// TwinCAT 3 PLC project PLC
// ProgramVersion: 3.1.4023.0
// libraries:
//   EfficientIO Communicator, * (EfficientIO)
//   EfficientIO ModbusTCP, * (EfficientIO)
//   Lynus Energy Basic, * (Lynus AG)
//   Lynus Persistent Data V1, * (Lynus AG)
//   Lynus Standards, * (Lynus AG)
//   Tc2_IoFunctions, * (Beckhoff Automation GmbH)
//   Tc2_ModbusRTU, * (Beckhoff Automation GmbH)
//   Tc2_ModbusSrv, * (Beckhoff Automation GmbH)
//   Tc2_SerialCom, * (Beckhoff Automation GmbH)
//   Tc2_Standard, * (Beckhoff Automation GmbH)
//   Tc2_System, * (Beckhoff Automation GmbH)
//   Tc2_Utilities, * (Beckhoff Automation GmbH)
//   Tc3_IotBase, * (Beckhoff Automation GmbH)
//   Tc3_Module, * (Beckhoff Automation GmbH)
// project tree:
//   DUTs/ ModbusRTURequest.TcDUT (not stored), struct_ADS_Barac.TcDUT (not stored)
//   / FastTask.TcTTO, MiddleTask.TcTTO, SlowTask.TcTTO
//   FB/ F_Convert_Reg_to_Real.TcPOU, MODBUS_RTU_Olymp.TcPOU
//   POUs/ prgBattery.TcPOU, prgComEffIO.TcPOU, prgCS.TcPOU, prgEM.TcPOU, prgEMS.TcPOU, prgHeatPump.TcPOU, prgPersistent.TcPOU, prgPV.TcPOU, prgRWEffIO.TcPOU (not stored), prgTemperature.TcPOU, prgVarEffIO.TcPOU
// real-time tasks:
//   TASK PlcTask: cycle T#10ms, priority 20, ADS port 350
//   TASK FastTask: cycle T#5ms, priority 19, ADS port 351
//   TASK MiddleTask: cycle T#10ms, priority 21, ADS port 352
//   TASK SlowTask: cycle T#20ms, priority 22, ADS port 353
// I/O:
//   DEVICE Gerät 2 (CX-BK)
//     Box 1 (CX-BK)
// variable links:
//   PLC/PLC Instance <-> Device 2 (CX-BK)/Box 1 (CX-BK)
//     FastTask Inputs/MODBUS_RTU_Olymp.fbModbusRtuMaster_KL6x22B.InData/D[{0..21}] <-> Term 6 (KL6041)/Channel 1/Data In {0..21}  (22 links)
//     FastTask Inputs/MODBUS_RTU_Olymp.fbModbusRtuMaster_KL6x22B.InData/Status <-> Term 6 (KL6041)/Channel 1/Status
//     FastTask Outputs/MODBUS_RTU_Olymp.fbModbusRtuMaster_KL6x22B.OutData/Ctrl <-> Term 6 (KL6041)/Channel 1/Ctrl
//     FastTask Outputs/MODBUS_RTU_Olymp.fbModbusRtuMaster_KL6x22B.OutData/D[{0..21}] <-> Term 6 (KL6041)/Channel 1/Data Out {0..21}  (22 links)
//     MiddleTask Inputs/prgEM.fbEM1.fbKL3403.byStateCH1 <-> Term 5 (KL3403)/Channel 1/Status
//     MiddleTask Inputs/prgEM.fbEM1.fbKL3403.byStateCH2 <-> Term 5 (KL3403)/Channel 2/Status
//     MiddleTask Inputs/prgEM.fbEM1.fbKL3403.byStateCH3 <-> Term 5 (KL3403)/Channel 3/Status
//     MiddleTask Inputs/prgEM.fbEM1.fbKL3403.iDataInCH1 <-> Term 5 (KL3403)/Channel 1/Daten Ein
//     MiddleTask Inputs/prgEM.fbEM1.fbKL3403.iDataInCH2 <-> Term 5 (KL3403)/Channel 2/Daten Ein
//     MiddleTask Inputs/prgEM.fbEM1.fbKL3403.iDataInCH3 <-> Term 5 (KL3403)/Channel 3/Daten Ein
//     MiddleTask Inputs/prgEM.fbKBusState.uiKBusState_OUT <-> Inputs/State
//     MiddleTask Inputs/prgTemperature.stInData_1/iDataIn <-> Term 4 (KL3204)/Channel 1/Daten Ein
//     MiddleTask Inputs/prgTemperature.stInData_2/iDataIn <-> Term 4 (KL3204)/Channel 2/Daten Ein
//     MiddleTask Inputs/prgTemperature.stInData_1/iState <-> Term 4 (KL3204)/Channel 1/Status
//     MiddleTask Inputs/prgTemperature.stInData_2/iState <-> Term 4 (KL3204)/Channel 2/Status
//     MiddleTask Outputs/prgEM.fbEM1.fbKL3403.byCntrCH1 <-> Term 5 (KL3403)/Channel 1/Kontrolle
//     MiddleTask Outputs/prgEM.fbEM1.fbKL3403.byCntrCH2 <-> Term 5 (KL3403)/Channel 2/Kontrolle
//     MiddleTask Outputs/prgEM.fbEM1.fbKL3403.byCntrCH3 <-> Term 5 (KL3403)/Channel 3/Kontrolle
//     MiddleTask Outputs/prgTemperature.bout_Boiler1_6kW <-> Term 3 (KL2408)/Channel 1/Ausgang
//     MiddleTask Outputs/prgTemperature.bout_Boiler2_10kW <-> Term 3 (KL2408)/Channel 2/Ausgang
//     MiddleTask Outputs/prgTemperature.stOutData_1/iCtrl <-> Term 4 (KL3204)/Channel 1/Kontrolle
//     MiddleTask Outputs/prgTemperature.stOutData_2/iCtrl <-> Term 4 (KL3204)/Channel 2/Kontrolle
//     MiddleTask Outputs/prgTemperature.stOutData_1/iDataOut <-> Term 4 (KL3204)/Channel 1/Daten Aus
//     MiddleTask Outputs/prgTemperature.stOutData_2/iDataOut <-> Term 4 (KL3204)/Channel 2/Daten Aus

CONFIGURATION PLC
    RESOURCE PLC ON TwinCAT3
        TASK FastTask(INTERVAL := T#5ms, PRIORITY := 19);
        TASK MiddleTask(INTERVAL := T#10ms, PRIORITY := 21);
        TASK SlowTask(INTERVAL := T#20ms, PRIORITY := 22);
        PROGRAM prgVarEffIO WITH FastTask : prgVarEffIO;
        PROGRAM prgRWEffIO WITH FastTask : prgRWEffIO;
        PROGRAM prgHeatPump WITH FastTask : prgHeatPump;
        PROGRAM prgEM WITH MiddleTask : prgEM;
        PROGRAM prgTemperature WITH MiddleTask : prgTemperature;
        PROGRAM prgPV WITH MiddleTask : prgPV;
        PROGRAM prgBattery WITH MiddleTask : prgBattery;
        PROGRAM prgEMS WITH MiddleTask : prgEMS;
        PROGRAM prgPersistent WITH MiddleTask : prgPersistent;
        PROGRAM prgCS WITH MiddleTask : prgCS;
        PROGRAM prgComEffIO WITH SlowTask : prgComEffIO;
    END_RESOURCE
END_CONFIGURATION

// ---- POUs/prgVarEffIO.TcPOU
PROGRAM prgVarEffIO
VAR
	fbVar		: FB_VarInfo_V3;
END_VAR

fbVar(
	bReadInfo:= , 
	eTMCFile:= eSelectTMCFile.eDontUseTMCFile, 
	eSavePositionTMCFile:= eSavePositionOnPLC.ePostionHardDisk, 
	udiCounterFoundVariables=> , 
	bError=> , 
	bBusy=> , 
	byProgress=> , 
	udiErrorCodeOut=> , 
	eErrorVarInfo_Out=> , 
	sVarWithError=> );

fbVar(
	bReadInfo:= , 
	eTMCFile:= eSelectTMCFile.eDontUseTMCFile, 
	eSavePositionTMCFile:= eSavePositionOnPLC.ePostionHardDisk, 
	udiCounterFoundVariables=> , 
	bError=> , 
	bBusy=> , 
	byProgress=> , 
	udiErrorCodeOut=> , 
	eErrorVarInfo_Out=> , 
	sVarWithError=> );
	
fbVar(
	bReadInfo:= , 
	eTMCFile:= eSelectTMCFile.eDontUseTMCFile, 
	eSavePositionTMCFile:= eSavePositionOnPLC.ePostionHardDisk, 
	udiCounterFoundVariables=> , 
	bError=> , 
	bBusy=> , 
	byProgress=> , 
	udiErrorCodeOut=> , 
	eErrorVarInfo_Out=> , 
	sVarWithError=> );

END_PROGRAM

// ---- POUs/prgHeatPump.TcPOU
PROGRAM prgHeatPump
VAR
	byte_OperationMode_H1: BYTE;							//{#lynus.ag#()}
	real_ComfortSetpoint_H1 :REAL;							//{#lynus.ag#()}
	real_ReducedSetpoint_H1: REAL;							//{#lynus.ag#()}
	real_HeatingCurveSlope_H1:REAL;							//{#lynus.ag#()}
	real_HeatingCurveDisplacement_H1: REAL;					//{#lynus.ag#()}
	real_RelativeRoomHumidity1_H1: REAL;	
	real_RoomTemperature1_H1 : REAL;
	real_RoomSetpoint1_H1 : REAL;
	real_FlowTemperature1_H1 : REAL;						//{#lynus.ag#()}
	real_FlowTemperatureSetpoint1_H1 : REAL;				//{#lynus.ag#()}
	m_RoomThermostat1_H1 : BOOL;							//{#lynus.ag#()}
	real_HeatOutput :REAL;									//{#lynus.ag#()}
	real_HeatInputSource :REAL;								//{#lynus.ag#()}
	real_PowerConsumption :REAL;							//{#lynus.ag#()}
	m_Heatingcircuit1_H1 : BOOL;							//{#lynus.ag#()}
	FB_DwordToWord :FB_CV_WORD_TO_DWORD;

	real_Outside_Temp : REAL;								//{#lynus.ag#()}
	real_Outside_Temp_min : REAL;							//{#lynus.ag#()}
	real_Outside_Temp_max : REAL;							//{#lynus.ag#()}
	real_Outside_Temp_attenuated : REAL;					//{#lynus.ag#()}
	real_Outside_Temp_composite : REAL;						//{#lynus.ag#()}

END_VAR

MODBUS_RTU_Olymp();

byte_OperationMode_H1 		:= 	WORD_TO_BYTE(Modbus_RTU_Olymp.structArrayModbusRTU[1].wArrayReceiveBuffer[0]);
real_ComfortSetpoint_H1		:= 	word_TO_REAL(Modbus_RTU_Olymp.structArrayModbusRTU[1].wArrayReceiveBuffer[1])/64;
real_ReducedSetpoint_H1		:= 	word_TO_REAL(Modbus_RTU_Olymp.structArrayModbusRTU[1].wArrayReceiveBuffer[2])/64;
real_HeatingCurveSlope_H1	:= 	WORD_TO_REAL(Modbus_RTU_Olymp.structArrayModbusRTU[1].wArrayReceiveBuffer[4])/50;
real_HeatingCurveDisplacement_H1:= 	WORD_TO_REAL(Modbus_RTU_Olymp.structArrayModbusRTU[1].wArrayReceiveBuffer[5])/64;
real_RelativeRoomHumidity1_H1:= 	word_TO_REAL(Modbus_RTU_Olymp.structArrayModbusRTU[1].wArrayReceiveBuffer[16])/1;
real_RoomTemperature1_H1	:= 	WORD_TO_REAL(Modbus_RTU_Olymp.structArrayModbusRTU[1].wArrayReceiveBuffer[18])/64;
real_RoomSetpoint1_H1		:= 	word_TO_REAL(Modbus_RTU_Olymp.structArrayModbusRTU[1].wArrayReceiveBuffer[20])/64;
real_FlowTemperature1_H1	:= 	word_TO_REAL(Modbus_RTU_Olymp.structArrayModbusRTU[2].wArrayReceiveBuffer[0])/64;
real_FlowTemperatureSetpoint1_H1:= 	WORD_TO_REAL(Modbus_RTU_Olymp.structArrayModbusRTU[2].wArrayReceiveBuffer[2])/64;
m_RoomThermostat1_H1		:= 	WORD_TO_BOOL(Modbus_RTU_Olymp.structArrayModbusRTU[2].wArrayReceiveBuffer[4]);
m_Heatingcircuit1_H1		:= 	WORD_TO_BOOL(Modbus_RTU_Olymp.structArrayModbusRTU[2].wArrayReceiveBuffer[9]);


FB_DwordToWord( 	wInputValue_1 := Modbus_RTU_Olymp.structArrayModbusRTU[5].wArrayReceiveBuffer[0],
					wInputValue_2 := Modbus_RTU_Olymp.structArrayModbusRTU[5].wArrayReceiveBuffer[1],
					eByteOrderForConvert :=,
					dwOutputValue =>);
real_HeatOutput				:= 	DWORD_TO_REAL(FB_DwordToWord.dwOutputValue)/100;

FB_DwordToWord( 	wInputValue_1 := Modbus_RTU_Olymp.structArrayModbusRTU[5].wArrayReceiveBuffer[3],
					wInputValue_2 := Modbus_RTU_Olymp.structArrayModbusRTU[5].wArrayReceiveBuffer[4],
					eByteOrderForConvert :=,
					dwOutputValue =>);
real_HeatInputSource			:= 	DWORD_TO_REAL(FB_DwordToWord.dwOutputValue)/100;
					
FB_DwordToWord( 	wInputValue_1 := Modbus_RTU_Olymp.structArrayModbusRTU[5].wArrayReceiveBuffer[6],
					wInputValue_2 := Modbus_RTU_Olymp.structArrayModbusRTU[5].wArrayReceiveBuffer[7],
					eByteOrderForConvert :=,
					dwOutputValue =>);
real_PowerConsumption			:= 	DWORD_TO_REAL(FB_DwordToWord.dwOutputValue)/100;



real_Outside_Temp 				:= INT_TO_REAL(WORD_TO_INT(Modbus_RTU_Olymp.structArrayModbusRTU[6].wArrayReceiveBuffer[4]))/64;
real_Outside_Temp_min			:= INT_TO_REAL(WORD_TO_INT(Modbus_RTU_Olymp.structArrayModbusRTU[6].wArrayReceiveBuffer[6]))/64;
real_Outside_Temp_max			:= INT_TO_REAL(WORD_TO_INT(Modbus_RTU_Olymp.structArrayModbusRTU[6].wArrayReceiveBuffer[7]))/64;
real_Outside_Temp_attenuated	:= INT_TO_REAL(WORD_TO_INT(Modbus_RTU_Olymp.structArrayModbusRTU[6].wArrayReceiveBuffer[8]))/64;
real_Outside_Temp_composite		:= INT_TO_REAL(WORD_TO_INT(Modbus_RTU_Olymp.structArrayModbusRTU[6].wArrayReceiveBuffer[9]))/64;

END_PROGRAM

// ---- FB/MODBUS_RTU_Olymp.TcPOU
PROGRAM MODBUS_RTU_Olymp

VAR_INPUT

END_VAR
VAR_OUTPUT
	dword_MB_Error		:ARRAY[1..3] OF DWORD;
END_VAR
VAR
//	fbModbusRtuMaster_KL6x22B: ModbusRtuMaster_KL6x22B;
	fbModbusRtuMaster_KL6x22B: ModbusRtuMasterV2_KL6x22B;
	fbConfigKL6041 : KL6Configuration;
	uintPollOrderCount: UINT;
	mBusy: BOOL;
	mError: BOOL;
	mStart: BOOL;
	udintMemoryDestAddress: UDINT;
	udintBytesReceived: UDINT;
	intState: INT:=0;
	timerT1: TON;
	timeWaitT1: TIME:=T#500MS;
	timeWaitT2: TIME:=T#500MS;
	timeNoRxTimeout:	TIME:=T#2S;
	timerT2: TON;

	fb_F_TRIG1: F_TRIG;
	timerTimeout: TON;
	mError_Rx: BOOL;
	udintErrorID: MODBUS_ERRORS;
	byteClientSlaveID: BYTE;
	uintNoOfWords: UINT;
	uintStartAddress: UINT;
	dw_Mask: DWORD;
	dw_Mask_Not: DWORD;
	uint_TestPollOrder: UINT;
	mTestMode: BOOL;
	mInit_Done: BOOL;
	
	structArrayModbusRTU	:ARRAY[1..60] OF ModbusRTURequest;
	uintMaxModbusRTUOrders: UINT;
	mExecute: BOOL;
	int_Handshake: ComHandshake_t:=4;
	mode: ComSerialLineMode_t:=3;
	byte_DataBits: BYTE:=8;
	i: UINT;
END_VAR

(*
The function block "ModbusRtuMaster_KL6x22B" has 22 bytes where it communicates with the plc
software. These 22 bytes have to be assigned to the hardware device (for example KL/EL6021) in the
system manager plus the control and status byte.
If devices with less then 22 bytes are used, the other function blocks have to be used (for 5 bytes for example).
*)

(*
IF fbModbusRtuMaster_KL6x22B.MBmaster.TimeoutTON.Q=TRUE AND mTimeOUT_Qold=FALSE THEN mTimeOUT_Q_Rising; END_IF
mTimeOUT_Qold:=fbModbusRtuMaster_KL6x22B.MBmaster.TimeoutTON.Q;
*)

fb_F_TRIG1(CLK:=mBusy);

CASE intState OF

0: 	(* reset the start bit *)
	mStart:=FALSE;
	IF mInit_Done AND NOT fbConfigKL6041.Busy THEN 
		intState:=10;
		mExecute:=FALSE;		
	ELSE
		INIT();
		mExecute:=TRUE;		// necessary to write the communication parameters to the KL terminal. only necessary once if the terminal is brand new
	END_IF
10:
	(* set next poll order *)
	uintPollOrderCount:=uintPollOrderCount+1; (* next slave *)
	WHILE NOT structArrayModbusRTU[uintPollOrderCount].mRequestActive DO
		uintPollOrderCount:=uintPollOrderCount+1; (* next slave *)
	END_WHILE
	
	(* trouble shooting *)
	IF mTestMode THEN
		uintPollOrderCount:=uint_TestPollOrder; (* next slave *)
	END_IF
	
	IF uintPollOrderCount > uintMaxModbusRTUOrders OR uintPollOrderCount<1 THEN
		uintPollOrderCount:=1;
	END_IF

	udintMemoryDestAddress:=ADR(structArrayModbusRTU[uintPollOrderCount].wArrayReceiveBuffer[0]);
	structArrayModbusRTU[uintPollOrderCount].udintBytesReceived:=0;
	mStart:=TRUE;
	timerTimeout.IN:=TRUE;
	intState:=20;

20: (* wait for busy falling or time out *)
	IF fb_F_TRIG1.Q OR timerTimeout.Q THEN

		(* check answer time *)
		structArrayModbusRTU[uintPollOrderCount].timeTimeForRequest:=timerTimeout.ET;

		(* reset timer *)
		timerTimeout.IN:=FALSE;

		(* reset start bit *)
		mStart:=FALSE;

		(* save number of bytes received *)
		structArrayModbusRTU[uintPollOrderCount].udintBytesReceived:=udintBytesReceived;
		udintBytesReceived:=0;

		(* Error Detection *)
		IF timerTimeout.Q THEN
			mError_Rx:=TRUE;
			structArrayModbusRTU[uintPollOrderCount].udintErrorID:=9998;
			structArrayModbusRTU[uintPollOrderCount].strErrorMessage:='Timeout';
		ELSIF structArrayModbusRTU[uintPollOrderCount].udintBytesReceived=0 AND structArrayModbusRTU[uintPollOrderCount].uintNoOfWords>0 THEN
			mError_Rx:=TRUE;
			structArrayModbusRTU[uintPollOrderCount].udintErrorID:=9999;
			structArrayModbusRTU[uintPollOrderCount].strErrorMessage:='0 bytes received';
		ELSIF fbModbusRtuMaster_KL6x22B.Error THEN
			mError_Rx:=TRUE;
			structArrayModbusRTU[uintPollOrderCount].udintErrorID:=udintErrorID;
//			structArrayModbusRTU[uintPollOrderCount].strErrorMessage:=F_ADSERRORTEXT(structArrayModbusRTU[uintPollOrderCount].udintErrorID);
		ELSE
			mError_Rx:=FALSE;
			structArrayModbusRTU[uintPollOrderCount].udintErrorID:=0;
			structArrayModbusRTU[uintPollOrderCount].strErrorMessage:='';
		END_IF


		IF mError_Rx THEN
			structArrayModbusRTU[uintPollOrderCount].udintCommErrorCounter:=structArrayModbusRTU[uintPollOrderCount].udintCommErrorCounter+1;
		ELSIF structArrayModbusRTU[uintPollOrderCount].udintBytesReceived>0 THEN (* Rev 3 *)
			structArrayModbusRTU[uintPollOrderCount].udintCommSuccessCounter:=structArrayModbusRTU[uintPollOrderCount].udintCommSuccessCounter+1;
		END_IF

		structArrayModbusRTU[uintPollOrderCount].timerOKTimer.IN:=NOT mError_Rx;
		structArrayModbusRTU[uintPollOrderCount].timerErrorTimer.IN:=mError_Rx;

		dw_Mask:=1;
		dw_Mask:=SHL(dw_Mask,(structArrayModbusRTU[uintPollOrderCount].intDeviceNumber));
		dw_Mask_Not:=NOT dw_Mask;
		
		IF structArrayModbusRTU[uintPollOrderCount].timerErrorTimer.Q THEN
			structArrayModbusRTU[uintPollOrderCount].mError:=TRUE;
			IF structArrayModbusRTU[uintPollOrderCount].intDeviceClass>=1 AND structArrayModbusRTU[uintPollOrderCount].intDeviceClass<=3 THEN
				dword_MB_Error[structArrayModbusRTU[uintPollOrderCount].intDeviceClass]:=dword_MB_Error[structArrayModbusRTU[uintPollOrderCount].intDeviceClass] OR dw_Mask;
			END_IF
		END_IF

		IF structArrayModbusRTU[uintPollOrderCount].timerOKTimer.Q THEN
			structArrayModbusRTU[uintPollOrderCount].mError:=FALSE;
			IF structArrayModbusRTU[uintPollOrderCount].intDeviceClass>=1 AND structArrayModbusRTU[uintPollOrderCount].intDeviceClass<=3 THEN
				dword_MB_Error[structArrayModbusRTU[uintPollOrderCount].intDeviceClass]:=dword_MB_Error[structArrayModbusRTU[uintPollOrderCount].intDeviceClass] AND dw_Mask_Not;
			END_IF
		END_IF

		(* clear buffer *)
		IF mError_Rx THEN
			MEMSET(destAddr:=udintMemoryDestAddress,fillByte:=0,130);
		END_IF

		(* set next state *)
		intState:=30;
	END_IF

30:		(* wait *)
		timerT1(IN:=TRUE);
		IF timerT1.Q THEN
			timerT1(IN:=FALSE);
			intState:=0; (* back to start *)
		END_IF

END_CASE

(* Timer calls *)
structArrayModbusRTU[uintPollOrderCount].timerErrorTimer(PT:=timeNoRxTimeout);
structArrayModbusRTU[uintPollOrderCount].timerOKTimer(PT:=T#2S);
timerT1(PT:=timeWaitT1);
timerT2(PT:=timeWaitT2);
timerTimeout(PT:=timeNoRxTimeout+timeWaitT1);


(* Timers *)
structArrayModbusRTU[uintPollOrderCount].timerErrorTimer.PT:=T#5S;
structArrayModbusRTU[uintPollOrderCount].timerOKTimer.PT:=T#5S;


//fbModbusRtuMaster_KL6x22B.ReadInputRegs(
fbModbusRtuMaster_KL6x22B.ReadRegs(
	UnitID:= structArrayModbusRTU[uintPollOrderCount].byteClientSlaveID, 
	Quantity:= structArrayModbusRTU[uintPollOrderCount].uintNoOfWords, 
	MBAddr:= structArrayModbusRTU[uintPollOrderCount].uintStartAddress , 
	cbLength:= 2*structArrayModbusRTU[uintPollOrderCount].uintNoOfWords,
	pMemoryAddr:= udintMemoryDestAddress, 
	AuxQuantity:= , 
	AuxMBAddr:= , 
	AuxcbLength:= , 
	pAuxMemoryAddr:= , 
	Execute:= mStart, 
	Timeout:= T#1S, 
	BUSY=> mBusy, 
	Error=> mError, 
	ErrorId=> udintErrorID, 
	cbRead=> udintBytesReceived);
	
(*fbModbusRtuMaster_KL6x22B.ReadRegs(
	UnitID		:=structArrayModbusRTU[uintPollOrderCount].byteClientSlaveID,
	Quantity	:=structArrayModbusRTU[uintPollOrderCount].uintNoOfWords,
	MBAddr		:=structArrayModbusRTU[uintPollOrderCount].uintStartAddress,
	cbLength	:=2*structArrayModbusRTU[uintPollOrderCount].uintNoOfWords,
	pMemoryAddr	:=udintMemoryDestAddress,
	Execute		:=mStart,
	Timeout		:=t#1s,
	BUSY		=>mBusy,
	Error		=>mError,
	ErrorId		=>udintErrorID,
	cbRead		=>udintBytesReceived
);
*)
(*
(*fbModbusRtuMaster_KL6x22B.ReadInputRegs(
*)
fbModbusRtuMaster_KL6x22B.ReadInputRegs(
	UnitID		:=structArrayModbusRTU[uintPollOrderCount].byteClientSlaveID,
	Quantity	:=structArrayModbusRTU[uintPollOrderCount].uintNoOfWords,
	MBAddr		:=structArrayModbusRTU[uintPollOrderCount].uintStartAddress,
	cbLength	:=2*structArrayModbusRTU[uintPollOrderCount].uintNoOfWords,
	pMemoryAddr	:=udintMemoryDestAddress,
	Execute		:=mStart,
	Timeout		:=t#1s,
	BUSY		=>mBusy,
	Error		=>mError,
	ErrorId		=>udintErrorID,
	cbRead		=>udintBytesReceived
);
*)
// necessary for KL6041 to wirte the com settings
fbConfigKL6041(
	Execute 		:= mExecute,
	Mode 			:= mode,
	Baudrate 		:= 19200,
	NoDatabits 		:= byte_DataBits,
	Parity 			:= 1,
	Stopbits 		:= 1,
	Handshake  		:= int_Handshake,
	ContinousMode 	:= FALSE,
	pComIn 			:= ADR(fbModbusRtuMaster_KL6x22B.InData),
	pComOut 		:= ADR(fbModbusRtuMaster_KL6x22B.OutData),
	SizeComIn 		:= SIZEOF(fbModbusRtuMaster_KL6x22B.InData)
);

ACTION INIT:


i:=1;
(* Poll 1 Heating circuit 1 *)
structArrayModbusRTU[i].byteClientSlaveID:=1;
structArrayModbusRTU[i].uintStartAddress:=1024;
structArrayModbusRTU[i].uintNoOfWords:=22;
structArrayModbusRTU[i].mRequestActive:=TRUE;

(* Poll 2 Heating Circuit 1 *)
i:=i+1;
structArrayModbusRTU[i].byteClientSlaveID:=1;
structArrayModbusRTU[i].uintStartAddress:=1046;
structArrayModbusRTU[i].uintNoOfWords:=22;
structArrayModbusRTU[i].mRequestActive:=TRUE;

(* Poll 3 Heating Circuit 1 *)
i:=i+1;
structArrayModbusRTU[i].byteClientSlaveID:=1;
structArrayModbusRTU[i].uintStartAddress:=1068;
structArrayModbusRTU[i].uintNoOfWords:=22;
structArrayModbusRTU[i].mRequestActive:=TRUE;

(* Poll 4 Heating Circuit 1 *)
i:=i+1;
structArrayModbusRTU[i].byteClientSlaveID:=1;
structArrayModbusRTU[i].uintStartAddress:=1090;
structArrayModbusRTU[i].uintNoOfWords:=2;
structArrayModbusRTU[i].mRequestActive:=TRUE;

(* Poll 5 Power*)
i:=i+1;
structArrayModbusRTU[i].byteClientSlaveID:=1;
structArrayModbusRTU[i].uintStartAddress:=20823;
structArrayModbusRTU[i].uintNoOfWords:=11;
structArrayModbusRTU[i].mRequestActive:=TRUE;

(* Poll 6 outside Temp*)
i:=i+1;
structArrayModbusRTU[i].byteClientSlaveID:=1;
structArrayModbusRTU[i].uintStartAddress:=35847;
structArrayModbusRTU[i].uintNoOfWords:=11;
structArrayModbusRTU[i].mRequestActive:=TRUE;



uintMaxModbusRTUOrders:=i;
mInit_Done:=TRUE;
END_ACTION

END_PROGRAM

// ---- POUs/prgEM.TcPOU
PROGRAM prgEM
VAR
	fbKBusState		: FB_K_Bus_State;
	fbEM1			: FB_EM_Beckhoff_KL3403;
	lrPower_Grid		: LREAL;						//{#lynus.ag#()}
	lrPower_Grid_L1		: LREAL;						//{#lynus.ag#()}
	lrPower_Grid_L2		: LREAL;						//{#lynus.ag#()}
	lrPower_Grid_L3		: LREAL;						//{#lynus.ag#()}
	lrCurrent_Grid_L1	: LREAL;						//{#lynus.ag#()}
	lrCurrent_Grid_L2	: LREAL;						//{#lynus.ag#()}
	lrCurrent_Grid_L3	: LREAL;						//{#lynus.ag#()}
	lrPower_House		: LREAL;						//{#lynus.ag#()}
	lrVoltage_Grid_L1N	: LREAL;						//{#lynus.ag#()}
	lrVoltage_Grid_L2N	: LREAL;						//{#lynus.ag#()}
	lrVoltage_Grid_L3N	: LREAL;						//{#lynus.ag#()}
	lrVoltage_Grid_L1L2	: LREAL;						//{#lynus.ag#()}
	lrVoltage_Grid_L2L3	: LREAL;						//{#lynus.ag#()}
	lrVoltage_Grid_L3L1	: LREAL;						//{#lynus.ag#()}
	x:int;
	fbGrid						: FB_Grid_Power;
	fbGridCounter				: FB_EnergyCounter;
	bEnableHouse		: BOOL:=TRUE;					//{#lynus.ag#()}
	bHouseEnabled		: BOOL:=TRUE;					//{#lynus.ag#()}
END_VAR
VAR PERSISTENT
	rSizeGridConn				: REAL;									//{#lynus.ag#()}
	lrCounterGridProd			: LREAL;								//{#lynus.ag#()}
	lrCounterGridCons			: LREAL;								//{#lynus.ag#()}
END_VAR


fbKBusState(	uiKBusState_OUT=> , 
				b_Kbus_notOk=> , 
				word_ErrorCount=> );
//The mapping OF THIS FUNCTION must be linked with the KL3403 in the E/A Part
// KEBA CS
fbEM1(
	bEnable:= true, 
	bChannel1Invers:= FALSE,				//Invert power data when transformer are mounted upside down
	bChannel2Invers:= FALSE,			
	bChannel3Invers:= FALSE,
	uiCurrentTransformerRatioL1:= 100, //Transformer ratio on the secondary side
	uiCurrentTransformerRatioL2:= 100, 
	uiCurrentTransformerRatioL3:= 100, 
	uiKBusState_IN:= fbKBusState.uiKBusState_OUT, 
	stDataEMPower=> , 
	stDataEMCounter=> , 
	stDataEMPowerRealTime=> , 
	stDataEMCounterRealTime=> , 
	diNrOfEM_OUT=> );
lrPower_Grid := fbEM1.stDataEMPower.lrPowerTotal;
lrPower_Grid_L1 := fbEM1.stDataEMPower.lrPowerL1;
lrPower_Grid_L2 := fbEM1.stDataEMPower.lrPowerL2;
lrPower_Grid_L3 := fbEM1.stDataEMPower.lrPowerL3;
lrCurrent_Grid_L1 := fbEM1.stDataEMPowerRealTime.lrCurrentL1;
lrCurrent_Grid_L2 := fbEM1.stDataEMPowerRealTime.lrCurrentL2;
lrCurrent_Grid_L3 := fbEM1.stDataEMPowerRealTime.lrCurrentL3;
lrVoltage_Grid_L1N:= fbEM1.stDataEMPowerRealTime.lrVoltageL1N;
lrVoltage_Grid_L2N:= fbEM1.stDataEMPowerRealTime.lrVoltageL2N;
lrVoltage_Grid_L3N:= fbEM1.stDataEMPowerRealTime.lrVoltageL3N;
lrVoltage_Grid_L1L2:= fbEM1.stDataEMPowerRealTime.lrVoltageL1L2;
lrVoltage_Grid_L2L3:= fbEM1.stDataEMPowerRealTime.lrVoltageL2L3;
lrVoltage_Grid_L3L1:= fbEM1.stDataEMPowerRealTime.lrVoltageL3L1;

lrPower_House := lrPower_Grid + prgPV.lrPowerPV + prgBattery.lrPowerBattery - prgTemperature.lr_Power_Heating1_6kW - prgTemperature.lr_Power_Heating2_10kW;

IF prgCS.lrPower <22 THEN 		// not sure if the MB readout is correct. 
	lrPower_House := lrPower_House - prgCS.lrPower;
END_IF
lrPower_House := MAX(0,lrPower_House);

fbGrid(
	bEnable:= TRUE, 
	diNrOfEMS_IN:= prgEMS.fbEMS.diNrOfEMS_OUT, 
	diNrOfEM_IN_Grid:= 	prgEM.fbEM1.diNrOfEM_OUT,		
	rSizeGridConn:= rSizeGridConn, 
	stDataGrid=> , 
	diNrOfGrid_OUT=> );
	
// EnergyCounter
fbGridCounter(
	byActiveTariff:= 1, 
	lrPowerInput:= lrPower_Grid, 
	lrTotalCounterEnergy_Consumption=> , 
	lrTotalCounterEnergy_Production=> , 
	lrCounterEnergyT1_Consumption=> , 
	lrCounterEnergyT2_Consumption=> , 
	lrCounterEnergyT1_Production=> , 
	lrCounterEnergyT2_Production=> );

END_PROGRAM

// ---- POUs/prgPV.TcPOU
PROGRAM prgPV
VAR PERSISTENT
END_VAR
VAR
	fbPV_1					: FB_Symo_PV_Inverter_FLOAT_1_DM_1_Inverter;
	fbPV_2					: FB_Symo_PV_Inverter_FLOAT_1_DM_1_Inverter;
	fbPVCounter				: FB_EnergyCounter;
	fbPVCounter_1				: FB_EnergyCounter;
	fbPVCounter_2				: FB_EnergyCounter;
	lrPowerPV				: LREAL;				//{#lynus.ag#()}
	byErrorWarningPV		: BYTE;					//{#lynus.ag#()}
	
	// extend or reduce amount of PV Inverters
	lrPowerPV_1				: LREAL;				//{#lynus.ag#()}
	lrPowerPV_2				: LREAL;				//{#lynus.ag#()}
	lrPower					: LREAL;				//{#lynus.ag#()}
	
END_VAR
VAR PERSISTENT
	lrCounterPV				: LREAL;				//{#lynus.ag#()}
	lrCounterPV_1			: LREAL;				//{#lynus.ag#()}
	lrCounterPV_2			: LREAL;				//{#lynus.ag#()}
	str_IP_PV1				: STRING(15):= '10.11.90.101';
	str_IP_PV2				: STRING(15):= '192.168.1.102';
	
END_VAR

fbPV_1(
	bEnable:= TRUE, 
	sIPAdress:= str_IP_PV1 , 
	byUnitID_Inverter:= , 
	stDataSymo10=> , 
	stDataEMPower_PV=> , 
	stDataEMCounter_PV=> , 
	diNrOfEM_OUT_PV=> );

fbPV_2(
	bEnable:= TRUE, 
	sIPAdress:= str_IP_PV2 , 
	byUnitID_Inverter:= , 
	stDataSymo10=> , 
	stDataEMPower_PV=> , 
	stDataEMCounter_PV=> , 
	diNrOfEM_OUT_PV=> );


	
lrPowerPV_1 := fbPV_1.stDataEMPower_PV.lrPowerTotal;
lrPowerPV_2 := fbPV_2.stDataEMPower_PV.lrPowerTotal;



lrPowerPV := lrPowerPV_1 + lrPowerPV_2;

// EnergyCounter
fbPVCounter(
	byActiveTariff:= 1, 
	lrPowerInput:= 0 - lrPowerPV, 
	lrTotalCounterEnergy_Consumption=> , 
	lrTotalCounterEnergy_Production=> , 
	lrCounterEnergyT1_Consumption=> , 
	lrCounterEnergyT2_Consumption=> , 
	lrCounterEnergyT1_Production=> , 
	lrCounterEnergyT2_Production=> );
	
IF fbPVCounter.lrTotalCounterEnergy_Production > lrCounterPV THEN  	
	lrCounterPV := fbPVCounter.lrTotalCounterEnergy_Production;
END_IF
// EnergyCounter
fbPVCounter_1(
	byActiveTariff:= 1, 
	lrPowerInput:= 0 - lrPowerPV_1, 
	lrTotalCounterEnergy_Consumption=> , 
	lrTotalCounterEnergy_Production=> , 
	lrCounterEnergyT1_Consumption=> , 
	lrCounterEnergyT2_Consumption=> , 
	lrCounterEnergyT1_Production=> , 
	lrCounterEnergyT2_Production=> );
	
IF fbPVCounter_1.lrTotalCounterEnergy_Production > lrCounterPV_1 THEN  	
	lrCounterPV_1 := fbPVCounter_1.lrTotalCounterEnergy_Production;
END_IF
// EnergyCounter
fbPVCounter_2(
	byActiveTariff:= 1, 
	lrPowerInput:= 0 - lrPowerPV_2, 
	lrTotalCounterEnergy_Consumption=> , 
	lrTotalCounterEnergy_Production=> , 
	lrCounterEnergyT1_Consumption=> , 
	lrCounterEnergyT2_Consumption=> , 
	lrCounterEnergyT1_Production=> , 
	lrCounterEnergyT2_Production=> );
	
IF fbPVCounter_2.lrTotalCounterEnergy_Production > lrCounterPV_2 THEN  	
	lrCounterPV_2 := fbPVCounter_2.lrTotalCounterEnergy_Production;
END_IF

END_PROGRAM

// ---- POUs/prgBattery.TcPOU
PROGRAM prgBattery
VAR PERSISTENT
	bEnableBattery				: BOOL:= true;					//{#lynus.ag#()}
	byPrioBattery				: BYTE;							//{#lynus.ag#()}
	lrMaxCapacityBattery		: LREAL;						//{#lynus.ag#()}
	lrCounterBattProd			: LREAL;						//{#lynus.ag#()}
	lrCounterBattCons			: LREAL;						//{#lynus.ag#()}
	str_IP						: STRING(15):='10.11.90.180';

END_VAR
VAR
	fbBattery					: FB_Xelectrix_Powerbox_v2;
	fbBattCounter				: FB_EnergyCounter;
	bIsEnabledBattery			: BOOL;							//{#lynus.ag#()}
	bResetBattery				: BOOL;							//{#lynus.ag#()}
	bSResetBattery				: BOOL;							//{#lynus.ag#()}
	byErrorWarningBattery		: BYTE;							//{#lynus.ag#()}
	dwSOCBattery				: DWORD;						//{#lynus.ag#()}
	rTargetPowerBattery			: REAL;							//{#lynus.ag#()}
	lrPowerBattery				: LREAL;						//{#lynus.ag#()}
	lrActualCapacityBattery		: LREAL;						//{#lynus.ag#()}
	byBatteryModbusError		: BOOL;							//{#lynus.ag#()}
	lrBatteryCons				: LREAL;						//{#lynus.ag#()}
	lrBatteryProd				: LREAL;						//{#lynus.ag#()}
	mtest						: BOOL;
	x: REAL;
	byBatteryIslandOperation	: BOOL;							//{#lynus.ag#()}
	byBatteryBypassOperation	: BOOL;							//{#lynus.ag#()}
	lrPowerGridBattery			: LREAL;						//{#lynus.ag#()}
END_VAR

IF mtest THEN
	Lynus_Standards.GVL_Energy.stDataOfBatteryInverters[1,1].rTargetPowerEMS:=x;
END_IF
fbBattery(
	bEnable:= bEnableBattery, 
	bActivateControl:=TRUE , 
	byUnitID:= 1, 
	byPriority:= byPrioBattery, 
	diNrOfEMS_IN:= prgEMS.fbEMS.diNrOfEMS_OUT, 
	lrMaxCapacityBattery:= lrMaxCapacityBattery, 
	sIPAdress:= str_IP, 						// modify IP Adress
	bReset:= bResetBattery, 
	m_ManualSetpointEnable:= , 
	i_SetpointPower_Manual_kW:= , 
	m_ManualChargeDischargeMax:= , 
	r_MaxChargePower_W:= , 
	r_MaxDischargePower_W:= , 
	m_go_to_online:= , 
	m_go_to_bypass:= , 
	stDataXelectrix=> , 
	stDataBatt=> , 
	stDataBattInverter=> , 
	stDataEMPower_Grid=> , 
	stDataEMCounter_Grid=> , 
	diNrOfBatt_OUT=> , 
	diNrOfBattInverter_OUT=> , 
	diNrOfEM_OUT_Grid=> , 
	lrMaxCapacityBattery_OUT=> , 
	iSetpointPower_Info=> , 
	dw_BatterySOC_notZero=> );
//Out
bIsEnabledBattery := fbBattery.stDataBatt.bEnabled;
bSResetBattery := fbBattery.stDataBattInverter.bStateReset;
dwSOCBattery := fbBattery.dw_BatterySOC_notZero;
rTargetPowerBattery := fbBattery.stDataBattInverter.rTargetPower;
lrPowerBattery := fbBattery.stDataBatt.lrPower;
lrActualCapacityBattery := fbBattery.lrMaxCapacityBattery_OUT;	
byErrorWarningBattery := fbBattery.stDataBatt.byErrorWarning;
byBatteryModbusError := fbBattery.stDataXelectrix.eErrorState = 1;
lrBatteryCons := fbBattery.stDataBatt.lrPowerConsumption;
lrBatteryProd := fbBattery.stDataBatt.lrPowerProduction;				
lrPowerGridBattery := 	fbBattery.stDataEMPower_Grid.lrPowerTotal;
					
// EnergyCounter
fbBattCounter(
	byActiveTariff:= 1, 
	lrPowerInput:= lrPowerBattery, 
	lrTotalCounterEnergy_Consumption=> , 
	lrTotalCounterEnergy_Production=> , 
	lrCounterEnergyT1_Consumption=> , 
	lrCounterEnergyT2_Consumption=> , 
	lrCounterEnergyT1_Production=> , 
	lrCounterEnergyT2_Production=> );
	
IF fbBattCounter.lrTotalCounterEnergy_Production > lrCounterBattProd THEN  	
	lrCounterBattProd := fbBattCounter.lrTotalCounterEnergy_Production;
END_IF

IF fbBattCounter.lrTotalCounterEnergy_Consumption > lrCounterBattCons THEN  	
	lrCounterBattCons := fbBattCounter.lrTotalCounterEnergy_Consumption;
END_IF

byBatteryIslandOperation := fbBattery.stDataXelectrix.eGridState=2;
byBatteryBypassOperation := NOT (fbBattery.stDataXelectrix.eBatteryState=4 OR fbBattery.stDataXelectrix.eBatteryState=5);

END_PROGRAM

// ---- POUs/prgEMS.TcPOU
PROGRAM prgEMS
VAR PERSISTENT
	byMaxDepthOfDischrgEPO		: BYTE;							//{#lynus.ag#()}
	byPrioMinChrgBattSOCInEPO	: BYTE;							//{#lynus.ag#()}
	byResChrgfromGridToBatt		: BYTE;							//{#lynus.ag#()}
	byResChrgfromGridToBatt_Controlled		: BYTE;							//{#lynus.ag#()}
	byReserveSOCEPO				: BYTE;							//{#lynus.ag#()}
	uiUpdateTime				: UINT;							//{#lynus.ag#()}
	bEnableEMS					: BOOL;							//{#lynus.ag#()}
	bAllowChrgFromGrid			: BOOL;							//{#lynus.ag#()}
	rMainFuseCSEMS				: REAL;							//{#lynus.ag#()}
	iOperationModeEMS			: INT;							//{#lynus.ag#()}
END_VAR
VAR
	fbEMS						: FB_EMS;
	bIsEnableEMS				: BOOL;							//{#lynus.ag#()}
	bStateAllowChrgFromGrid		: BOOL;							//{#lynus.ag#()}
	bHPActivate					: BOOL;							//{#lynus.ag#()}
	bControllingState			: BOOL;							//{#lynus.ag#()}
	iMessageEMS					: INT;							//{#lynus.ag#()}
	rHeartbeatEMS				: REAL;							//{#lynus.ag#()}
	rErrorWarningEMS			: REAL;							//{#lynus.ag#()}
	rReadyEMS					: REAL;							//{#lynus.ag#()}
	rNewBatteryPowerEMS			: REAL;							//{#lynus.ag#()}
END_VAR

fbEMS.stSetupEMS.bAllowChrgFromGrid := bAllowChrgFromGrid;
fbEMS.stSetupEMS.byMaxDepthOfDischrgEPO := byMaxDepthOfDischrgEPO;
fbEMS.stSetupEMS.byPrioMinChrgBattSOCInEPO := byPrioMinChrgBattSOCInEPO;
fbEMS.stSetupEMS.byReserveSOCEPO := byReserveSOCEPO;
fbEMS.stSetupEMS.rSizeMainFuseCS := rMainFuseCSEMS;
fbEMS.stSetupEMS.uiUpdateTime := uiUpdateTime;

IF iOperationModeEMS = 0 THEN fbEMS.eOperationMode := E_OperatingMode_EMS.eAllOff;
ELSIF iOperationModeEMS = 1 THEN fbEMS.eOperationMode := E_OperatingMode_EMS.eSelfConsumption;	
ELSIF iOperationModeEMS = 2 THEN fbEMS.eOperationMode := E_OperatingMode_EMS.ePeakLoadCapping;
ELSIF iOperationModeEMS = 3 THEN fbEMS.eOperationMode := E_OperatingMode_EMS.eLoadManagement;			
END_IF

fbEMS(
	bEnable						:= bEnableEMS, 
	diNrOfEM_IN_ECS				:= , 
	stSetupEMS					:= , 
	eOperationMode				:= , 
	eSpeedModeBackendController	:= E_SpeedModeBackendController_EMS.eFast, 
	eSpeedModeLocalController	:= E_SpeedModeLocalController_EMS.eFast,
	bActivateHP					:= bHPActivate, 
	bControllingState			:= TRUE, // bControllingState, 
	rHeartbeat					:= rHeartbeatEMS, 
	rErrorWarning				:= rErrorWarningEMS, 
	rEnergyOptReady				:= rReadyEMS, 
	rNewBattPower				:= rNewBatteryPowerEMS, 
	b_ZeroPowerRegulation		:=,
	b_EnableBatteryChargingControl	:= FALSE,
	b_StartReleaseBatteryCharging 	:= ,
	b_StopReleaseBatteryCharging 	:= ,
	rMaxBattChargingPower			:= 100,
	rPeakDetectionforCalculation 	:= 3,	// was original 3, caused issues that load management not caluculeted. see EMS line 313
	
	eMessageEMS				=> iMessageEMS, 
	bStateEnable			=> bIsEnableEMS, 
	bStateAllowChrgFromGrid	=> bStateAllowChrgFromGrid, 
	bMissingPowerData		=> , 
	bSurplusAvailable		=> , 
	byProgress				=> , 
	uiState_OUT				=> , 
	diNrOfEMS_OUT			=> , 
	arrMinPrioReached		=> , 
	arrMaxPrioReached		=> ,
	b_TimeBasedReleaseChargingBattery => );

END_PROGRAM

// ---- POUs/prgTemperature.TcPOU
PROGRAM prgTemperature
VAR
// Kanal 1
	fb_Config_1			: FB_KL320xConfig;
	stInData_1   		AT%I*		: ST_KL320xInData;
	stOutData_1		  	AT%Q*		: ST_KL320xOutData;
// Kanal 2
	fb_Config_2			: FB_KL320xConfig;
	stInData_2   		AT%I*		: ST_KL320xInData;
	stOutData_2  		AT%Q*		: ST_KL320xOutData;
	lrTemperature_Top		: LREAL;						//{#lynus.ag#()}
	lrTemperature_Bottom	: LREAL;						//{#lynus.ag#()}
// do für heizstäbe

	bout_Boiler1_6kW		AT%Q*: BOOL;
	bout_Boiler2_10kW		AT%Q*: BOOL;
	b_Boiler_Heizstab6kW_ein		: BOOL;						//{#lynus.ag#()}
	b_Boiler_Heizstab10kW_ein		: BOOL;						//{#lynus.ag#()}
	lr_Power_Heating1_6kW			: LREAL;						//{#lynus.ag#()}
	lr_Power_Heating2_10kW			: LREAL;						//{#lynus.ag#()}


END_VAR

bout_Boiler1_6kW 	:= 	b_Boiler_Heizstab6kW_ein;
bout_Boiler2_10kW	:= 	b_Boiler_Heizstab10kW_ein;

lr_Power_Heating1_6kw 	:= SEL(bout_Boiler1_6kW,0,6);
lr_Power_Heating2_10kW 	:= SEL(bout_Boiler2_10kW,0,10);



	
fb_Config_1(
	bConfigurate:= , 
	bReadConfig:= , 
	iSetSensorType:= , 
	tTimeout:= , 
	bBusy=> , 
	bError=> , 
	iErrorId=> , 
	iState=> , 
	iDataIn=> , 
	iTerminalType=> , 
	iSpecialType=> , 
	iFirmwareVersion=> , 
	sDescription=> , 
	sSensorType=> , 
	bTwoWiredConnection=> , 
	stInData:= stInData_1, 
	stOutData:= stOutData_1);
lrTemperature_Top := INT_TO_LREAL(fb_Config_1.iDataIn)/10;
	
fb_Config_2(
	bConfigurate:= , 
	bReadConfig:= , 
	iSetSensorType:= , 
	tTimeout:= , 
	bBusy=> , 
	bError=> , 
	iErrorId=> , 
	iState=> , 
	iDataIn=> , 
	iTerminalType=> , 
	iSpecialType=> , 
	iFirmwareVersion=> , 
	sDescription=> , 
	sSensorType=> , 
	bTwoWiredConnection=> , 
	stInData:= stInData_2, 
	stOutData:= stOutData_2);
lrTemperature_Bottom := INT_TO_LREAL(fb_Config_2.iDataIn)/10;

END_PROGRAM

// ---- POUs/prgCS.TcPOU
PROGRAM prgCS
VAR
	bSManualyOn				: BOOL;												//{#lynus.ag#()}
	bEnabled				: BOOL;												//{#lynus.ag#()}
	bySManualyTargetPower	: BYTE;												//{#lynus.ag#()}
	bySMinPowerECS			: BYTE;												//{#lynus.ag#()}
	byErrorWarning			: BYTE;												//{#lynus.ag#()}
	lrPowerTotal			: LREAL;											//{#lynus.ag#()}
	lrPower					: LREAL;											//{#lynus.ag#()}
	rChargingTimeInMin		: REAL;												//{#lynus.ag#()}
	rTargetPower			: REAL;												//{#lynus.ag#()}
	wState					: WORD;												//{#lynus.ag#()}
	lrEnergySession			: LREAL;											//{#lynus.ag#()}
	lrTotalEnergy			: LREAL;											//{#lynus.ag#()}
	bCarConnected			: BOOL;												//{#lynus.ag#()}
	FB_MB_FC4		:FB_ModBus_2Registers_FC4;
	str_ip: STRING(15):='192.168.1.155';
END_VAR
VAR PERSISTENT
	bEnable					: BOOL;												//{#lynus.ag#()}
	bManualyOn				: BOOL;												//{#lynus.ag#()}
	byMinPower				: BYTE;												//{#lynus.ag#()}
	byManualyTargetPower	: BYTE;												//{#lynus.ag#()}
	byPrio					: BYTE;												//{#lynus.ag#()}
	bySOCEnable				: BYTE;												//{#lynus.ag#()}
	bySOCDisable			: BYTE;												//{#lynus.ag#()}
	rMaxPower				: REAL;												//{#lynus.ag#()}
	
END_VAR

// temp for reading out the charging power	
FB_MB_FC4(
	m_Enable:= TRUE, 
	str_IPAdress:= '192.168.1.155', 
	w_Adress:= 782, 
	int_Divider:= 1, 
	n_UnitID:= 255, 
	m_Float32Conversion:= , 
	m_LittleEndian:= , 
	m_PollSuccessful=> , 
	r_ReceivedValue=> , 
	udint_Error_ID=> );
	
lrPower := 	REAL_TO_LREAL(FB_MB_FC4.r_ReceivedValue)/1000;
lrPowerTotal := lrPower;

END_PROGRAM

// ---- POUs/prgPersistent.TcPOU
PROGRAM prgPersistent
VAR
	fbUSV		: FB_WritePersistentData_CX81xx;
	fb_Reboot		: NT_reboot;
	m_Reboot		: BOOL:=FALSE;
END_VAR

fbUSV(
	eSaveModeData:= eUSVSaveMode.eSaveWhenPowerfail, 
	bLoadPersistentDataOk=> , 
	bPowerFailDetect=> , 
	bError=> , 
	bySaveProcess=> , 
	dwStorageLast24h=> , 
	udiErrorCode=> );

	
fb_Reboot(	netid := '',
			delay := 2,
			start := m_Reboot);

END_PROGRAM

// ---- POUs/prgComEffIO.TcPOU
PROGRAM prgComEffIO
VAR
	fbCom		: FB_MqttCommunicator_v3;
//	fbCom2		: FB_MqttCommunicator;


	byte_array : ARRAY[0..1023] OF BYTE;
	struct_transfer	: struct_ADS_Barac;

	mSize_to_Big: BOOL;
	uint_size: UINT;
END_VAR

fbCom(
	bConnect:= TRUE, 
	strAuthkey := 'BMS99299754422',
	sUserName:= 'c4f8afbf-2040-4517-95e7-ed7f0d999242' , 		
	sUserPassword:= '14fc1314-6e6e-40a6-914d-101b441e17be',
	eSavePositionCertificate:= eSavePositionOnPLC.ePostionHardDisk, 
	bConnected=> , 
	bError=> , 
	hrErrorCode=> , 
	eConnectionState=> , 
	eErrorMessage_Out=> );
	
	(*old
		sUserName:= 'f8baf60b-d8e6-4d61-9ab1-e27d2122d4fe' , 		
	sUserPassword:= 'c431e8a4-3506-458b-8e70-7e5db8a7022f',
*)

// copy values to struct
struct_transfer.int_liveCount 				:= struct_transfer.int_liveCount+1;
struct_transfer.bIsEnableEMS			  	:= prgEMS.bIsEnableEMS;
struct_transfer.bStateAllowChrgFromGrid		:= prgEMS.bStateAllowChrgFromGrid;
struct_transfer.rHeartbeatEMS				:= prgEMS.rHeartbeatEMS;
struct_transfer.rErrorWarningEMS			:= prgEMS.rErrorWarningEMS;
struct_transfer.rReadyEMS					:= prgEMS.rReadyEMS;
struct_transfer.iOperationModeEMS			:= prgEMS.iOperationModeEMS;
struct_transfer.byMaxDepthOfDischrgEPO		:= prgEMS.byMaxDepthOfDischrgEPO;
struct_transfer.byReserveSOCEPO				:= prgEMS.byReserveSOCEPO;
struct_transfer.byPrioMinChrgBattSOCInEPO	:= prgEMS.byPrioMinChrgBattSOCInEPO;
struct_transfer.byResChrgfromGridToBatt		:= prgEMS.byResChrgfromGridToBatt;
struct_transfer.uiUpdateTime				:= prgEMS.uiUpdateTime;
struct_transfer.bEnableEMS					:= prgEMS.bEnableEMS;
struct_transfer.rNewBatteryPowerEMS			:= prgEMS.rNewBatteryPowerEMS;
struct_transfer.bHPActivate					:= prgEMS.bHPActivate;
struct_transfer.bAllowChrgFromGrid			:= prgEMS.bAllowChrgFromGrid;
struct_transfer.bControllingState			:= prgEMS.bControllingState;
struct_transfer.rMainFuseCSEMS				:= prgEMS.rMainFuseCSEMS;
struct_transfer.lrPowerPV_1					:= prgPV.lrPowerPV_1;
struct_transfer.lrPowerPV_2					:= prgPV.lrPowerPV_2;
struct_transfer.lrPower_Grid				:= prgEM.lrPower_Grid;
struct_transfer.rSizeGridConn				:= prgEM.rSizeGridConn;
struct_transfer.byBatteryIslandOperation	:= prgBattery.byBatteryIslandOperation;
struct_transfer.lrPowerBattery				:= prgBattery.lrPowerBattery;
struct_transfer.dwSOCBattery				:= prgBattery.dwSOCBattery;
struct_transfer.rTargetPowerBattery			:= prgBattery.rTargetPowerBattery;
struct_transfer.bIsEnabledBattery			:= prgBattery.bIsEnabledBattery;
struct_transfer.bSResetBattery				:= prgBattery.bSResetBattery;
struct_transfer.lrActualCapacityBattery		:= prgBattery.lrActualCapacityBattery;
struct_transfer.lrMaxCapacityBattery		:= prgBattery.lrMaxCapacityBattery;
struct_transfer.byPrioBattery				:= prgBattery.byPrioBattery;
struct_transfer.bEnableBattery				:= prgBattery.bEnableBattery;
struct_transfer.bResetBattery				:= prgBattery.bResetBattery;
struct_transfer.byBatteryBypassOperation	:= prgBattery.byBatteryBypassOperation;
struct_transfer.lrPower_House				:= prgEM.lrPower_House;
struct_transfer.bEnableHouse				:= prgEM.bEnableHouse;
struct_transfer.bHouseEnabled				:= prgEM.bHouseEnabled;
struct_transfer.lrPowerGridBattery			:= prgBattery.lrPowerGridBattery;
struct_transfer.lrPower_Grid_L1				:= prgEM.lrPower_Grid_L1;
struct_transfer.lrPower_Grid_L2				:= prgEM.lrPower_Grid_L2;
struct_transfer.lrPower_Grid_L3				:= prgEM.lrPower_Grid_L3;
struct_transfer.lrCurrent_Grid_L1			:= prgEM.lrCurrent_Grid_L1 ;
struct_transfer.lrCurrent_Grid_L2			:= prgEM.lrCurrent_Grid_L2 ;
struct_transfer.lrCurrent_Grid_L3			:= prgEM.lrCurrent_Grid_L3 ;
struct_transfer.lrVoltage_Grid_L1N			:= prgEM.lrVoltage_Grid_L1N;
struct_transfer.lrVoltage_Grid_L2N			:= prgEM.lrVoltage_Grid_L2N;
struct_transfer.lrVoltage_Grid_L3N			:= prgEM.lrVoltage_Grid_L3N;
(*struct_transfer.		:= ;
struct_transfer.		:= ;
struct_transfer.		:= ;
struct_transfer.		:= ;
struct_transfer.		:= ;
struct_transfer.		:= ;
struct_transfer.		:= ;
struct_transfer.		:= ;
*)


// copy struct to byte array
IF SIZEOF(struct_transfer) > SIZEOF(byte_array) THEN
	memcpy(ADR(byte_array),ADR(struct_transfer),SIZEOF(byte_array));
	uint_size := SIZEOF(struct_transfer);
	mSize_to_Big := TRUE;
ELSE
	memcpy(ADR(byte_array),ADR(struct_transfer),SIZEOF(struct_transfer));
	mSize_to_Big := FALSE;
END_IF
uint_size := SIZEOF(struct_transfer);

END_PROGRAM

// ---- FB/F_Convert_Reg_to_Real.TcPOU
FUNCTION F_Convert_Reg_to_Real : REAL
VAR_INPUT
	word_in1:WORD;
	word_in2:WORD;
END_VAR
VAR
	word_in	:ARRAY[0..1] OF WORD;
END_VAR

word_in[0]:=word_in1;
word_in[1]:=word_in2;

memcpy(ADR(F_Convert_Reg_to_Real),ADR(word_in),SIZEOF(word_in));

END_FUNCTION
